FUNCTION_BLOCK FB_System_WDT_Sollwertscheck
VAR_IN_OUT
	Zustand		: ST_System_WDT_Zustand;
END_VAR
VAR_INPUT
	Steuerung	: ST_System_WDT_Steuerung;
END_VAR
VAR
END_VAR

(* Priorisierung Regelung_Modus *)
IF(Steuerung.Regelung_Modus.manu_Modus) THEN
	Zustand.Regelung_Modus := Steuerung.Regelung_Modus.manu;
ELSIF(Steuerung.Regelung_Modus.opti_Modus) THEN
	Zustand.Regelung_Modus := Steuerung.Regelung_Modus.opti;
ELSE
	Zustand.Regelung_Modus := Steuerung.Regelung_Modus.auto;
END_IF;
(* Priorisierung Regelung_Nachtabs *)
IF(Steuerung.Regelung_Nachtabs.manu_Modus) THEN
	Zustand.Regelung_Nachtabs := Steuerung.Regelung_Nachtabs.manu;
ELSIF(Steuerung.Regelung_Nachtabs.opti_Modus) THEN
	Zustand.Regelung_Nachtabs := Steuerung.Regelung_Nachtabs.opti;
ELSE
	Zustand.Regelung_Nachtabs := Steuerung.Regelung_Nachtabs.auto;
END_IF;
(* Priorisierung Regelung_Sollwert *)
IF(Steuerung.Regelung_Sollw.manu_Modus) THEN
	Zustand.Regelung_Sollw_Anford := Steuerung.Regelung_Sollw.manu;
ELSIF(Steuerung.Regelung_Sollw.opti_Modus) THEN
	Zustand.Regelung_Sollw_Anford := Steuerung.Regelung_Sollw.opti;
ELSE
	Zustand.Regelung_Sollw_Anford := Steuerung.Regelung_Sollw.auto;
END_IF;

Zustand.Regelung_Sollw	:=	Zustand.Regelung_Sollw_Anford;

END_FUNCTION_BLOCK

(* stored: Version 1.1.0.1, ProductVersion 3.1.4024.9
   POU FB_System_WDT_Sollwertscheck: Id {0835af0d-74f8-43e5-b45e-f068564aacdd}, SpecialFunc None *)
